// SIMATIC S7-200 SMART project (STEP 7-Micro/WIN SMART), CPU CR40

SYMBOL_TABLE 表格 1
CPU_输出_0         Q0.0     // 料仓电机
CPU_输出_1         Q0.1     // 回转气缸
CPU_输出_10        Q1.2     // 绿灯
CPU_输出_2         Q0.2     // 伸缩气缸
CPU_输出_3         Q0.3     // 升降气缸
CPU_输出_4         Q0.4     // 气动手抓
CPU_输出_8         Q1.0     // 红灯
CPU_输出_9         Q1.1     // 黄灯
CPU_输入_14        I1.6     // 工件检测
CPU_输入_15        I1.7     // 摆臂左限位
CPU_输入_16        I2.0     // 启动
CPU_输入_17        I2.1     // 暂停
CPU_输入_18        I2.2     // RES1
CPU_输入_19        I2.3     // 急停
CPU_输入_2         I0.2     // 摆臂右限位
CPU_输入_20        I2.4     // 料仓检测
CPU_输入_22        I2.6     // AUT
CPU_输入_3         I0.3     // 气缸伸出限位
CPU_输入_4         I0.4     // 气缸收回限位
CPU_输入_5         I0.5     // 上升限位
CPU_输入_6         I0.6     // 下降限位
CPU_输入_7         I0.7     // 工作夹检测
END_SYMBOL_TABLE

SYMBOL_TABLE 系统符号
Always_On        SM0.0    // 始终接通
First_Scan_On    SM0.1    // 仅在第一个扫描周期时接通
Clock_1s         SM0.5    // 针对 1 s 的周期时间，时钟脉冲接通 0.5 s，断开 0.5 s.
END_SYMBOL_TABLE

ORGANIZATION_BLOCK MAIN:OB1
TITLE=程序注释
BEGIN
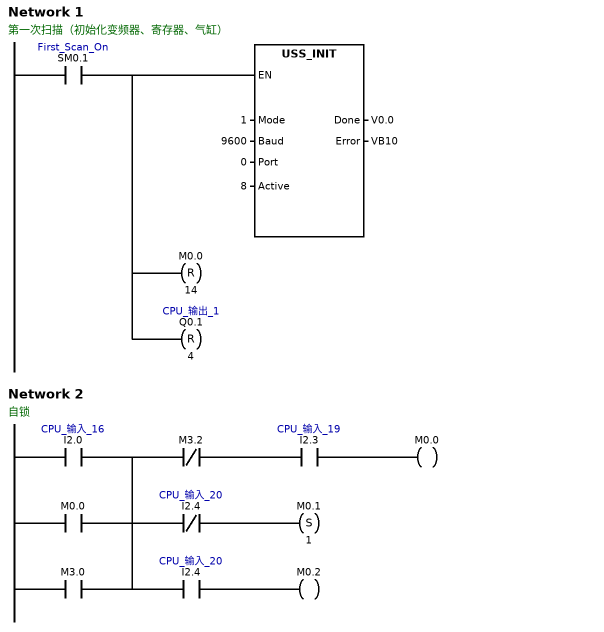
Network 1
// 第一次扫描（初始化变频器、寄存器、气缸）
LD     First_Scan_On:SM0.1
CALL   USS_INIT:SBR1, 1, 9600, 0, 8, V0.0, VB10
R      M0.0, 14
R      CPU_输出_1:Q0.1, 4
Network 2
// 自锁
LD     CPU_输入_16:I2.0
O      M0.0
O      M3.0
LPS
AN     M3.2
A      CPU_输入_19:I2.3
=      M0.0
LRD
AN     CPU_输入_20:I2.4
S      M0.1, 1
LPP
A      CPU_输入_20:I2.4
=      M0.2
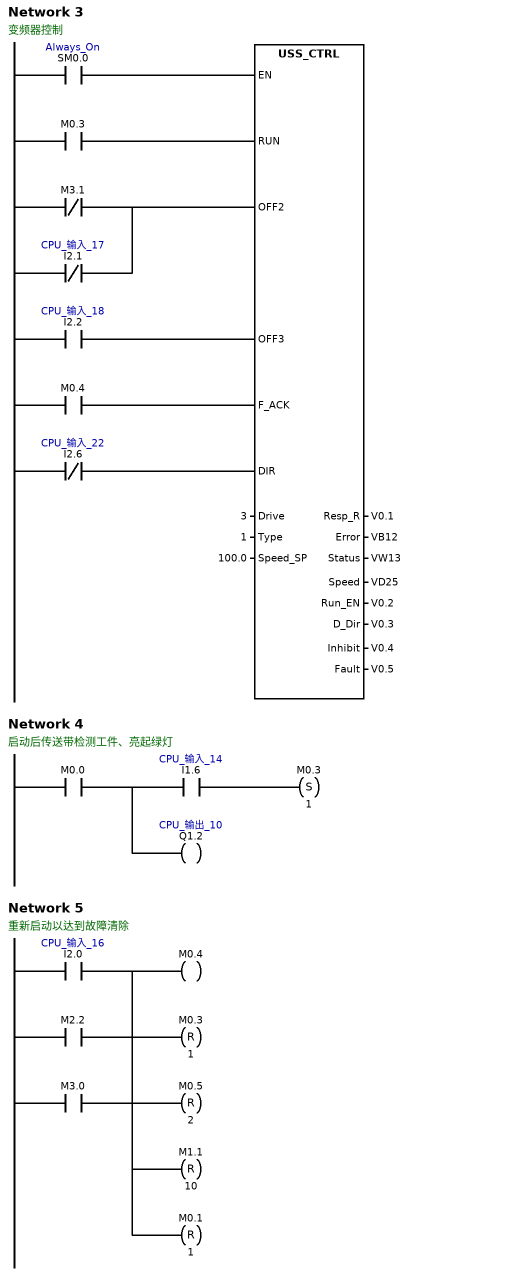
Network 3
// 变频器控制
LD     Always_On:SM0.0
=      L60.0
LD     M0.3
=      L63.7
LDN    M3.1
ON     CPU_输入_17:I2.1
=      L63.6
LD     CPU_输入_18:I2.2
=      L63.5
LD     M0.4
=      L63.4
LDN    CPU_输入_22:I2.6
=      L63.3
LD     L60.0
CALL   USS_CTRL:SBR5, L63.7, L63.6, L63.5, L63.4, L63.3, 3, 1, 100.0, V0.1, VB12, VW13, VD25, V0.2, V0.3, V0.4, V0.5
Network 4
// 启动后传送带检测工件、亮起绿灯
LD     M0.0
LPS
A      CPU_输入_14:I1.6
S      M0.3, 1
LPP
=      CPU_输出_10:Q1.2
Network 5
// 重新启动以达到故障清除
LD     CPU_输入_16:I2.0
O      M2.2
O      M3.0
=      M0.4
R      M0.3, 1
R      M0.5, 2
R      M1.1, 10
R      M0.1, 1
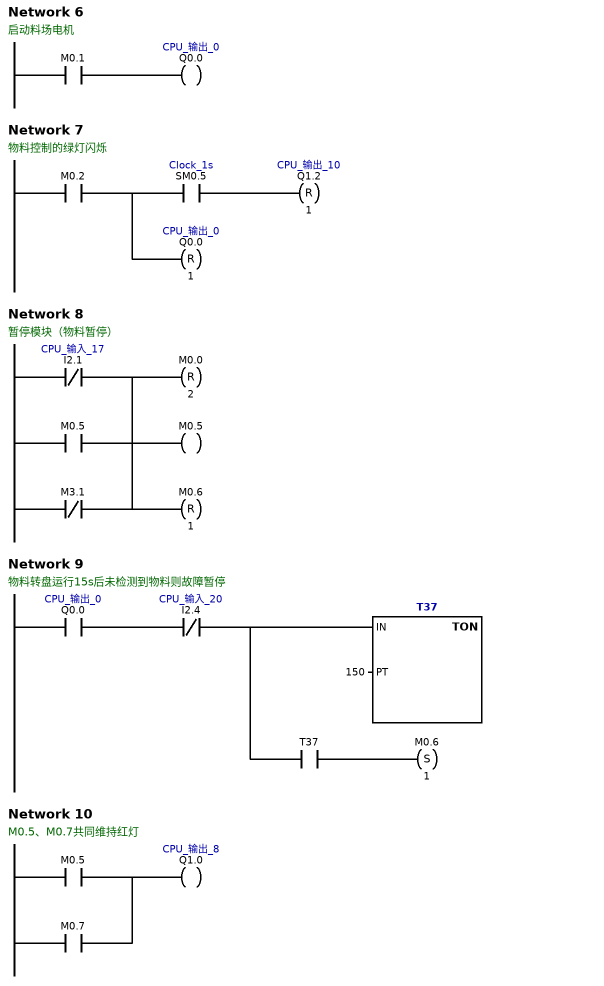
Network 6
// 启动料场电机
LD     M0.1
=      CPU_输出_0:Q0.0
Network 7
// 物料控制的绿灯闪烁
LD     M0.2
LPS
A      Clock_1s:SM0.5
R      CPU_输出_10:Q1.2, 1
LPP
R      CPU_输出_0:Q0.0, 1
Network 8
// 暂停模块（物料暂停）
LDN    CPU_输入_17:I2.1
O      M0.5
ON     M3.1
R      M0.0, 2
=      M0.5
R      M0.6, 1
Network 9
// 物料转盘运行15s后未检测到物料则故障暂停
LD     CPU_输出_0:Q0.0
AN     CPU_输入_20:I2.4
TON    T37, 150
A      T37
S      M0.6, 1
Network 10
// M0.5、M0.7共同维持红灯
LD     M0.5
O      M0.7
=      CPU_输出_8:Q1.0
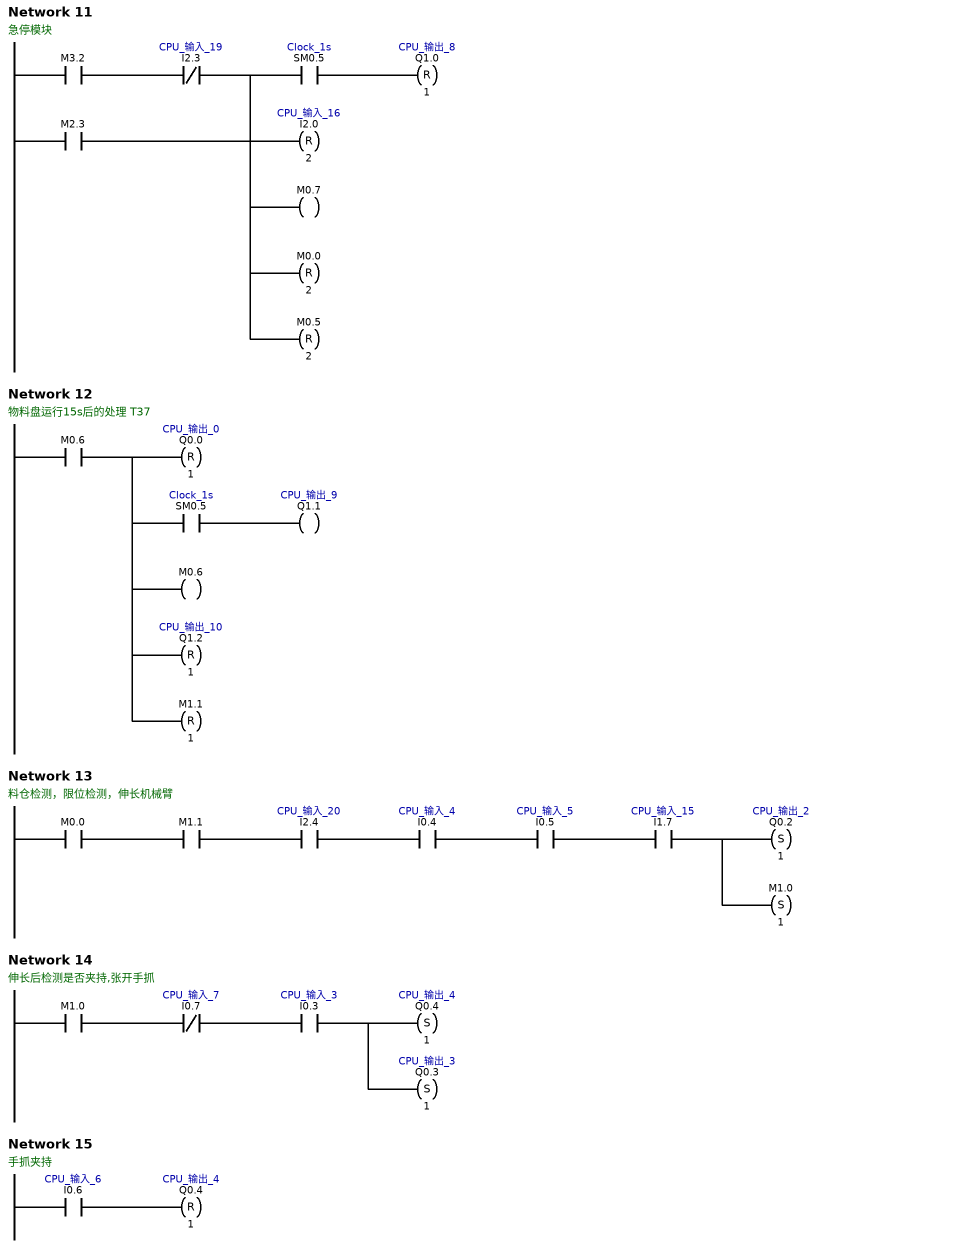
Network 11
// 急停模块
LD     M3.2
AN     CPU_输入_19:I2.3
O      M2.3
LPS
A      Clock_1s:SM0.5
R      CPU_输出_8:Q1.0, 1
LRD
R      CPU_输入_16:I2.0, 2
LRD
=      M0.7
LRD
R      M0.0, 2
LPP
R      M0.5, 2
Network 12
//  物料盘运行15s后的处理 T37
LD     M0.6
LPS
R      CPU_输出_0:Q0.0, 1
A      Clock_1s:SM0.5
=      CPU_输出_9:Q1.1
LRD
=      M0.6
LRD
R      CPU_输出_10:Q1.2, 1
LPP
R      M1.1, 1
Network 13
// 料仓检测，限位检测，伸长机械臂	
LD     M0.0
A      M1.1
A      CPU_输入_20:I2.4
A      CPU_输入_4:I0.4
A      CPU_输入_5:I0.5
A      CPU_输入_15:I1.7
S      CPU_输出_2:Q0.2, 1
S      M1.0, 1
Network 14
// 伸长后检测是否夹持,张开手抓
LD     M1.0
AN     CPU_输入_7:I0.7
A      CPU_输入_3:I0.3
S      CPU_输出_4:Q0.4, 1
S      CPU_输出_3:Q0.3, 1
Network 15
// 手抓夹持
LD     CPU_输入_6:I0.6
R      CPU_输出_4:Q0.4, 1
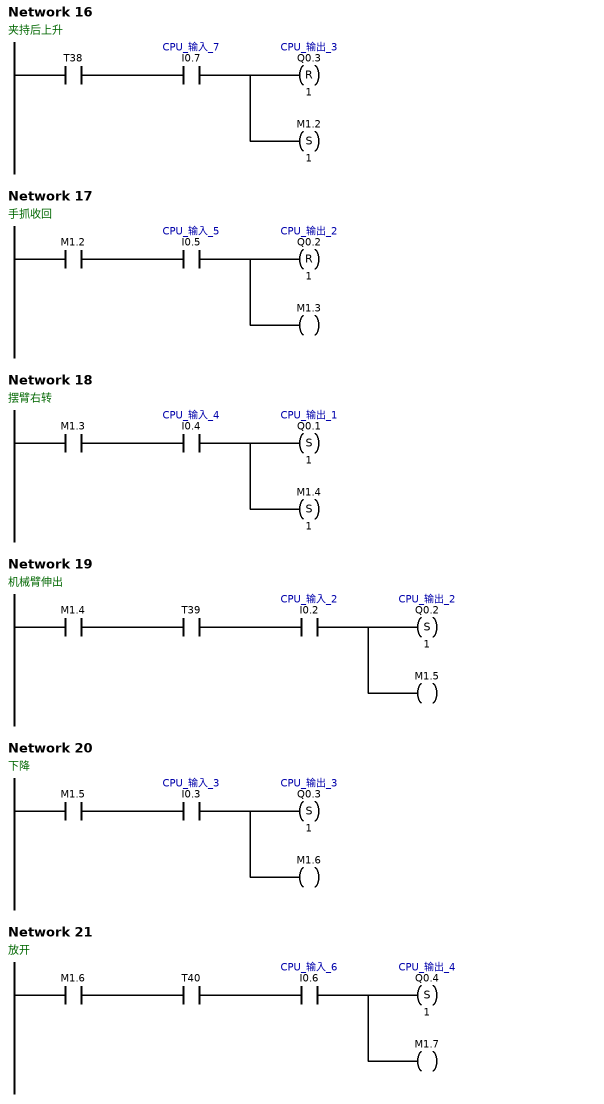
Network 16
// 夹持后上升
LD     T38
A      CPU_输入_7:I0.7
R      CPU_输出_3:Q0.3, 1
S      M1.2, 1
Network 17
// 手抓收回
LD     M1.2
A      CPU_输入_5:I0.5
R      CPU_输出_2:Q0.2, 1
=      M1.3
Network 18
// 摆臂右转
LD     M1.3
A      CPU_输入_4:I0.4
S      CPU_输出_1:Q0.1, 1
S      M1.4, 1
Network 19
// 机械臂伸出
LD     M1.4
A      T39
A      CPU_输入_2:I0.2
S      CPU_输出_2:Q0.2, 1
=      M1.5
Network 20
// 下降
LD     M1.5
A      CPU_输入_3:I0.3
S      CPU_输出_3:Q0.3, 1
=      M1.6
Network 21
// 放开
LD     M1.6
A      T40
A      CPU_输入_6:I0.6
S      CPU_输出_4:Q0.4, 1
=      M1.7
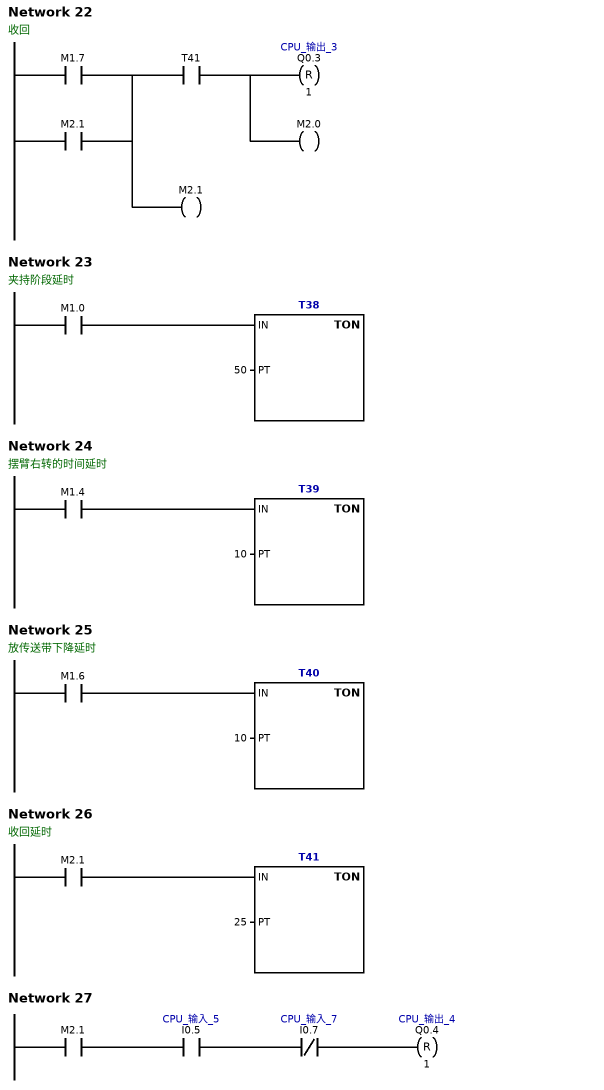
Network 22
// 收回
LD     M1.7
O      M2.1
LPS
A      T41
R      CPU_输出_3:Q0.3, 1
=      M2.0
LPP
=      M2.1
Network 23
// 夹持阶段延时
LD     M1.0
TON    T38, 50
Network 24
// 摆臂右转的时间延时
LD     M1.4
TON    T39, 10
Network 25
// 放传送带下降延时
LD     M1.6
TON    T40, 10
Network 26
// 收回延时
LD     M2.1
TON    T41, 25
Network 27
LD     M2.1
A      CPU_输入_5:I0.5
AN     CPU_输入_7:I0.7
R      CPU_输出_4:Q0.4, 1
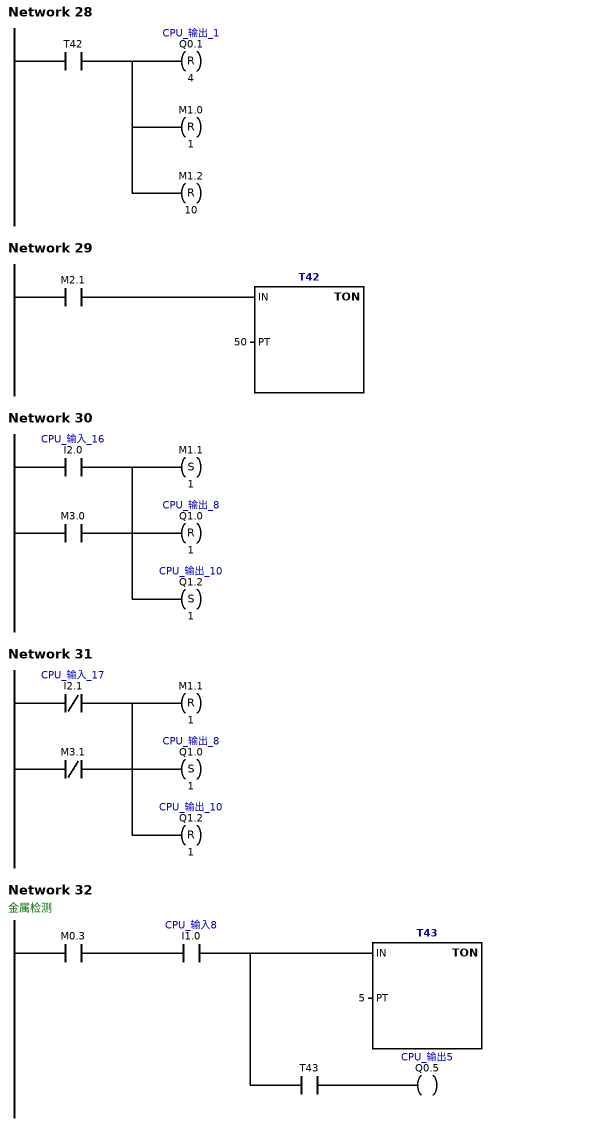
Network 28
LD     T42
R      CPU_输出_1:Q0.1, 4
R      M1.0, 1
R      M1.2, 10
Network 29
LD     M2.1
TON    T42, 50
Network 30
LD     CPU_输入_16:I2.0
O      M3.0
S      M1.1, 1
R      CPU_输出_8:Q1.0, 1
S      CPU_输出_10:Q1.2, 1
Network 31
LDN    CPU_输入_17:I2.1
ON     M3.1
R      M1.1, 1
S      CPU_输出_8:Q1.0, 1
R      CPU_输出_10:Q1.2, 1
Network 32
// 金属检测
LD     M0.3
A      CPU_输入8:I1.0
TON    T43, 5
A      T43
=      CPU_输出5:Q0.5
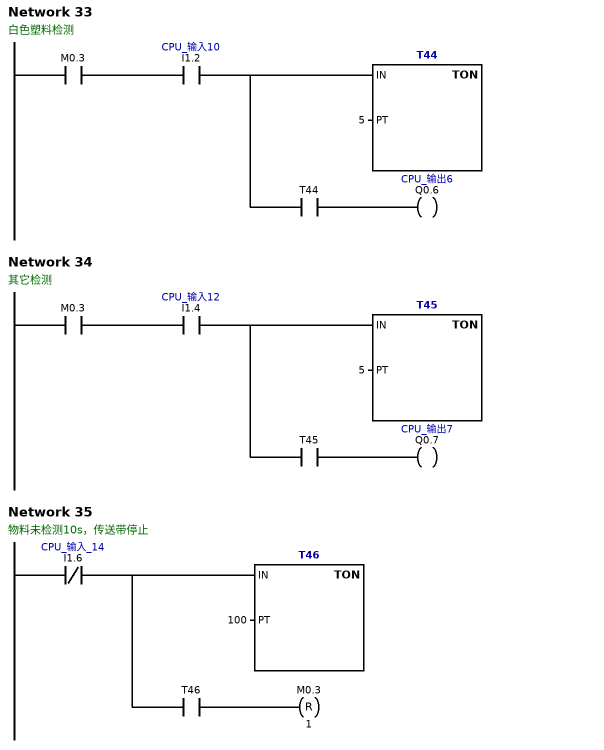
Network 33
// 白色塑料检测
LD     M0.3
A      CPU_输入10:I1.2
TON    T44, 5
A      T44
=      CPU_输出6:Q0.6
Network 34
// 其它检测
LD     M0.3
A      CPU_输入12:I1.4
TON    T45, 5
A      T45
=      CPU_输出7:Q0.7
Network 35
// 物料未检测10s，传送带停止
LDN    CPU_输入_14:I1.6
TON    T46, 100
A      T46
R      M0.3, 1
END_ORGANIZATION_BLOCK

// SBR1: protected block, not included

// SBR2: protected block, not included

// SBR3: protected block, not included

// SBR4: protected block, not included

// SBR5: protected block, not included

// INT1: protected block, not included
